// TwinCAT 3 PLC project PLC
// ProgramVersion: 3.1.4023.0
// libraries:
//   Tc2_Standard, * (Beckhoff Automation GmbH)
//   Tc2_System, * (Beckhoff Automation GmbH)
//   Tc3_Module, * (Beckhoff Automation GmbH)
// project tree:
//   GVLs/ DUT.TcDUT, G_task1.TcGVL, P_task1.TcPOU
//   / PlcTask.TcTTO
//   POUs/ MAIN.TcPOU
// real-time tasks:
//   TASK PlcTask: cycle T#10ms, priority 20, ADS port 350

CONFIGURATION PLC
    RESOURCE PLC ON TwinCAT3
        TASK PlcTask(INTERVAL := T#10ms, PRIORITY := 20);
        PROGRAM MAIN WITH PlcTask : MAIN;
    END_RESOURCE
END_CONFIGURATION

// ---- GVLs/DUT.TcDUT
{attribute 'qualified_only'}
{attribute 'strict'}
TYPE DUT :
(
	Sick := 1,
	Pilz := 2,
	Parker :=3,
 	Bosch := 4
);
END_TYPE

// ---- GVLs/G_task1.TcGVL
VAR_GLOBAL
	dtVariable: DATE_AND_TIME := DT#2020-04-04-05:31:19;
	dtTime : TIME := T#10S;
	sensor1 : DUT; 
	sensor2  : DUT;
	bStart : BOOL := TRUE;
	bQ : BOOL := TRUE;
	fbTon: TON:= (PT:=T#10S);
END_VAR

// ---- POUs/MAIN.TcPOU
PROGRAM MAIN
VAR
END_VAR

P_task1();

END_PROGRAM

// ---- GVLs/P_task1.TcPOU
PROGRAM P_task1
VAR
	pPointer: POINTER TO DATE_AND_TIME := ADR(dtVariable);
	nRef_Time: REFERENCE TO TIME REF=dtTime;
	aDates: ARRAY[1..4] OF DATE_AND_TIME := [DT#2023-02-07-00:00:00,DT#2023-02-08-00:00:00,DT#2023-02-09-00:00:00,DT#2023-02-10-00:00:00];
END_VAR

pPointer^:= DT#2023-04-04-05:31:19;
// nRef_Time:= T#1S;
aDates[3]:=DT#2023-02-25-00:00:00;
G_task1.sensor1:= DUT.Bosch;
G_task1.sensor2:= DUT.Parker;

fbTon(IN:= G_task1.bQ);

END_PROGRAM
